FUNCTION_BLOCK EL2652
VAR
	{attribute addProperty Name "WcState"}
	_wcState : WcStateBase;
	{attribute addProperty Name "Info data"}
	_infoData : InfoDataBase;
	_io : EL2xx2_Data;
END_VAR

PROPERTY IO : REFERENCE TO EL2xx2_Data
GET
IO REF= _io;
END_GET
END_PROPERTY

PROPERTY WcState : REFERENCE TO WcStateBase
GET
WcState REF= _wcState;
END_GET
END_PROPERTY

END_FUNCTION_BLOCK

(* stored: Version 1.1.0.1, ProductVersion 3.1.4024.9
   POU EL2652: Id {36a4ffc6-5c8e-0cdc-2dd8-157daad6a086}, SpecialFunc None
   Property IO: Id {25e0d1dc-845b-0525-0028-c39f9bfcb014}
   Get Get: Id {e632106c-1d0c-0f81-1c86-db29851a0928}
   Property WcState: Id {c52fe9a3-74ae-0a67-2bec-556cdefe2330}
   Get Get: Id {6eb53ca1-59bc-05ea-095c-819f8836a7ef} *)
